(* PLC project Unbenannt, Unbekannt Unbenannt 1 *)
(* stored: creationDateTime 2019-09-02T13:12:52, modificationDateTime 2019-09-02T13:50:06 *)

FUNCTION_BLOCK STACK_32
  VAR_INPUT
    DIN : DWORD;
    _E : BOOL := TRUE;
    RD : BOOL;
    WD : BOOL;
    RST : BOOL;
  END_VAR
  VAR_OUTPUT
    DOUT : DWORD;
    EMPTY : BOOL := TRUE;
    FULL : BOOL;
  END_VAR
  VAR
    pt : INT;
    stack : ARRAY[0..31] OF DWORD;
  END_VAR

            IF RST THEN

	(* asynchronous reset for the fifo *)

	pt := 0;

	EMPTY := TRUE;

	FULL := FALSE;

	Dout := DWORD#0;

ELSIF _E THEN

	IF NOT EMPTY AND RD THEN

		(* read one element *)

		pt := pt - 1;

		Dout := stack[pt];

		EMPTY := pt = 0;

		FULL := FALSE;

	END_IF;

	IF NOT FULL AND WD THEN

		(* write one element *)

		stack[pt] := Din;

		pt := pt + 1;

		FULL := pt > 31;

		EMPTY := FALSE;

	END_IF;

END_IF;


(* from OSCAT library; www.oscat.de  *)
          
END_FUNCTION_BLOCK

(* This is a increment function which increments the variable X by 1 and if N is reached, it begins with 0 instead of N again. *)
FUNCTION INC1 : INT
  VAR_INPUT
    X : INT;
    N : INT;
  END_VAR

            IF X >= N - 1 THEN
	INC1 := 0;
ELSE
	INC1 := X + 1;
END_IF;
(* from OSCAT library; www.oscat.de  *)
          
END_FUNCTION

FUNCTION_BLOCK FIFO_32
  VAR_INPUT
    DIN : DWORD;
    _E : BOOL := TRUE;
    RD : BOOL;
    WD : BOOL;
    RST : BOOL;
  END_VAR
  VAR_OUTPUT
    DOUT : DWORD;
    EMPTY : BOOL := TRUE;
    FULL : BOOL;
  END_VAR
  VAR
    fifo : ARRAY[0..31] OF DWORD;
    pr : INT;
    pw : INT;
  END_VAR

            IF RST THEN

	pw := pr;

	FULL := FALSE;

	EMPTY := TRUE;

	Dout := DWORD#0;

ELSIF _E THEN

	IF NOT EMPTY AND RD THEN

		Dout := fifo[pr];

		pr := INC1(pr,32);

		EMPTY := pr = pw;

		FULL := FALSE;

	END_IF;

	IF NOT FULL AND WD THEN

		fifo[pw] := Din;

		pw := INC1(pw,32);

		FULL := pw = pr;

		EMPTY := FALSE;

	END_IF;

END_IF;



(* from OSCAT library; www.oscat.de  *)
          
END_FUNCTION_BLOCK

PROGRAM program0
  VAR
    LocalVar0 : DINT;
    LocalVar1 : DINT;
    LocalVar2 : DINT;
  END_VAR

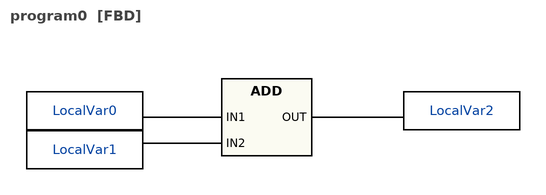
(* FBD diagram, written out as Structured Text *)
LocalVar2 := LocalVar0 + LocalVar1;
END_PROGRAM

FUNCTION_BLOCK FIFO_16
  VAR_INPUT
    DIN : DWORD;
    _E : BOOL := TRUE;
    RD : BOOL;
    WD : BOOL;
    RST : BOOL;
  END_VAR
  VAR_OUTPUT
    DOUT : DWORD;
    EMPTY : BOOL := TRUE;
    FULL : BOOL;
  END_VAR
  VAR
    fifo : ARRAY[0..15] OF DWORD;
    pr : INT;
    pw : INT;
  END_VAR

            IF RST THEN

	pw := pr;

	FULL := FALSE;

	EMPTY := TRUE;

	Dout := DWORD#0;

ELSIF _E THEN

	IF NOT EMPTY AND RD THEN

		Dout := fifo[pr];

		pr := INC1(pr,16);

		EMPTY := pr = pw;

		FULL := FALSE;

	END_IF;

	IF NOT FULL AND WD THEN

		fifo[pw] := Din;

		pw := INC1(pw,16);

		FULL := pw = pr;

		EMPTY := FALSE;

	END_IF;

END_IF;


(* from OSCAT library; www.oscat.de  *)
          
END_FUNCTION_BLOCK

FUNCTION_BLOCK STACK_16
  VAR_INPUT
    DIN : DWORD;
    _E : BOOL := TRUE;
    RD : BOOL;
    WD : BOOL;
    RST : BOOL;
  END_VAR
  VAR_OUTPUT
    DOUT : DWORD;
    EMPTY : BOOL := TRUE;
    FULL : BOOL;
  END_VAR
  VAR
    pt : INT;
    stack : ARRAY[0..15] OF DWORD;
  END_VAR

            IF RST THEN

	(* asynchronous reset for the fifo *)

	pt := 0;

	EMPTY := TRUE;

	FULL := FALSE;

	Dout := DWORD#0;

ELSIF _E THEN

	IF NOT EMPTY AND RD THEN

		(* read one element *)

		pt := pt - 1;

		Dout := stack[pt];

		EMPTY := pt = 0;

		FULL := FALSE;

	END_IF;

	IF NOT FULL AND WD THEN

		(* write one element *)

		stack[pt] := Din;

		pt := pt + 1;

		FULL := pt > 15;

		EMPTY := FALSE;

	END_IF;

END_IF;


(* from OSCAT library; www.oscat.de  *)
          
END_FUNCTION_BLOCK

CONFIGURATION Config0
  RESOURCE Res0 ON PLC
    TASK task0(INTERVAL := T#20ms, PRIORITY := 0);
    PROGRAM instance0 WITH task0 : program0;
  END_RESOURCE
END_CONFIGURATION
